(* Schneider Machine Expert - Basic project Motor 3 fasa Delta Star 2, file version 1.7.0.0 *)
(* ProjectInformations: Name=New project *)

HARDWARE
  Cpu 0: TM221M16R/G
  EthernetConfiguration: NetworkName=M221, IpAllocationMode=FixedAddress, IpAddress=0.0.0.0, SubnetMask=0.0.0.0
  SerialLineConfiguration: Baud=Baud19200, Parity=ParityEven, DataBits=DataBits8, StopBits=StopBits1, PhysicalMedium=PhysicalMediumRs485, TransmissionMode=TransmissionModeModbusRtu, SlaveId=1, Addressing=SlaveAddressing
  MastTask: UsePeriodScanMode=false, PeriodScan=100
  FastTask: Period=255
  CpuBehavior: StartingMode=StartAsPreviousState, AutoSaveRamOnEeprom=true, WatchdogPeriod=250

SYMBOLS  (address, symbol, comment, settings)
  %TM0        "T1"  [Preset=15, Base=OneSecond]
  %I0.0       "PB1"
  %I0.1       "PB2"
  %Q0.0       "K1M"
  %Q0.1       "K2M"
  %Q0.2       "K3M"

POU New POU
  (* SectionNumber=1 *)

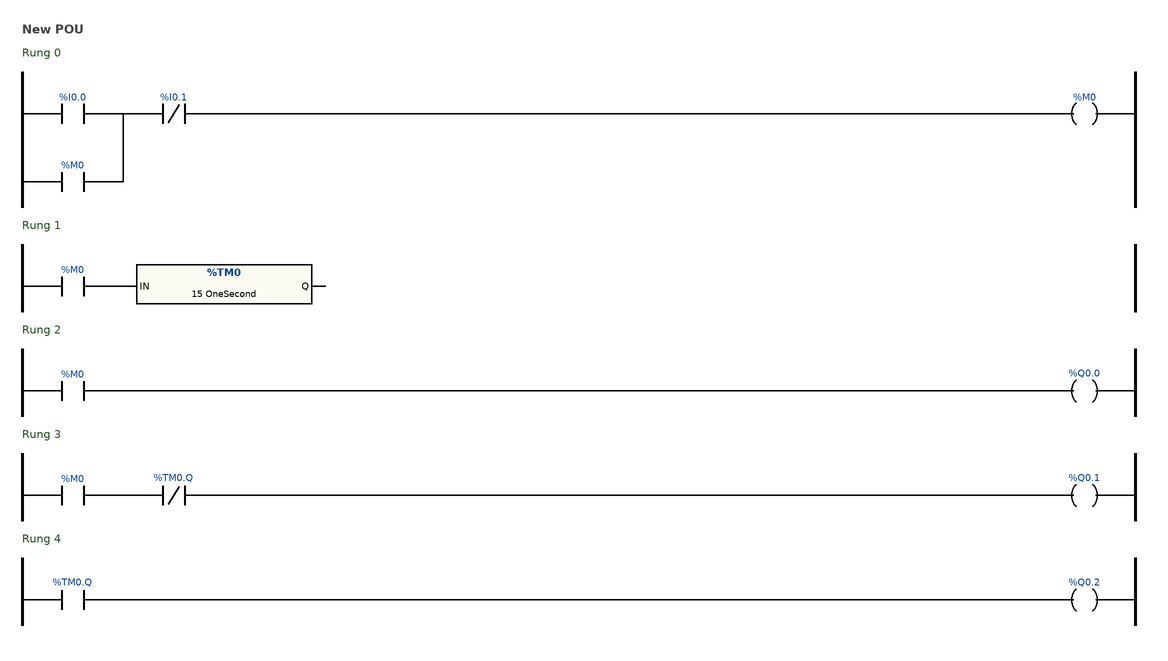

// Rung 0
  LD %I0.0
  OR %M0
  ANDN %I0.1
  ST %M0
  // as ST:
  //   %M0 := (%I0.0 OR %M0) AND NOT %I0.1;

// Rung 1
  BLK %TM0
  LD %M0
  IN
  END_BLK
  // as ST:
  //   %TM0(IN := %M0);

// Rung 2
  LD %M0
  ST %Q0.0
  // as ST:
  //   %Q0.0 := %M0;

// Rung 3
  LD %M0
  ANDN %TM0.Q
  ST %Q0.1
  // as ST:
  //   %Q0.1 := %M0 AND NOT %TM0.Q;

// Rung 4
  LD %TM0.Q
  ST %Q0.2
  // as ST:
  //   %Q0.2 := %TM0.Q;
